(* CODESYS project Command3.project

Project tree, tasks and I/O mapping:
  Device : CODESYS Control for Raspberry Pi SL, 3S - Smart Software Solutions GmbH, version 3.5.11.0
    application Application
      libraries: Standard, * (System); StringUtils, 3.5.11.0 (System); CoDeSys Memory Manager, 3.5.12.0 (3S - Smart Software Solutions GmbH)
      task Task (cyclic, interval t#20ms, priority 1) calls MAIN
      POUs/
        Commands/
          function block FB_SocketOffCommand [ST]: Execute, FB_init, Undo
          function block FB_AirConComfortCommand [ST]: Execute, FB_init, Undo
          function block FB_AirConStandbyCommand [ST]: Execute, FB_init, Undo
          function block FB_SocketOnCommand [ST]: Execute, FB_init, Undo
          function block FB_LampSetLevelCommand [ST]: Execute, FB_init, Undo
          function block FB_MusicPlayCommand [ST]: Execute, FB_init, Undo
          function block FB_MusicStopCommand [ST]: Undo, Execute, FB_init
          interface I_Command: Execute, Undo
        Receiver/
          function block FB_Socket [ST]: Active, Off, On
          function block FB_Lamp [ST]: SetLevel, Level
          function block FB_CDPlayer [ST]: Volume, SetTrack, SetVolume, Start, Stop, PlayerActive, Track
          function block FB_AirConditioning [ST]: Activate, Deactivate, SetTemperature, Activated, Temperature
        Invoker/
          function block FB_SwitchPanel [ST]: FB_init, SetCommand
        program MAIN [ST]
    SoftMotion General Axis Pool
    I²C
    SPI
    GPIOs_A_B : GPIOs A/B, 3S - Smart Software Solutions GmbH, version 3.5.11.0
        unmapped channels: digital inputs (GPIO0..GPIO31), digital outputs (GPIO0..GPIO31)
    Onewire
    Camera device
      <Empty>
*)

// Device/Application/POUs/MAIN
PROGRAM MAIN
VAR
	// Invoker
	fbSwitchPanel				: FB_SwitchPanel;
	
	// Receiver
	fbSocket					: FB_Socket;
	refSocket					: REFERENCE TO FB_Socket := fbSocket;	
	fbLamp						: FB_Lamp;
	refLamp						: REFERENCE TO FB_Lamp := fbLamp;	
	fbAirConditioning			: FB_AirConditioning;
	refAirConditioning			: REFERENCE TO FB_AirConditioning := fbAirConditioning;
	fbCDPlayer					: FB_CDPlayer;
	refCDPlayer					: REFERENCE TO FB_CDPlayer := fbCDPlayer;

	// Commands
	fbSocketOnCommand			: FB_SocketOnCommand(refSocket);
	fbSocketOffCommand			: FB_SocketOffCommand(refSocket);
	fbLampSetLevel100Command	: FB_LampSetLevelCommand(refLamp, 100);
	fbLampSetLevel0Command		: FB_LampSetLevelCommand(refLamp, 0);
	fbAirConComfortCommand		: FB_AirConComfortCommand(refAirConditioning);
	fbAirConStandbyCommand		: FB_AirConStandbyCommand(refAirConditioning);	
	fbMusicPlayCommand			: FB_MusicPlayCommand(refCDPlayer);
	fbMusicStopCommand			: FB_MusicStopCommand(refCDPlayer);
	bInit						      : BOOL := TRUE;	
END_VAR

IF bInit THEN
	fbSwitchPanel.SetCommand(1, fbSocketOnCommand);
	fbSwitchPanel.SetCommand(2, fbSocketOffCommand);
	fbSwitchPanel.SetCommand(3, fbLampSetLevel100Command);
	fbSwitchPanel.SetCommand(4, fbLampSetLevel0Command);
	fbSwitchPanel.SetCommand(5, fbAirConComfortCommand);
	fbSwitchPanel.SetCommand(6, fbAirConStandbyCommand);
	fbSwitchPanel.SetCommand(7, fbMusicPlayCommand);
	fbSwitchPanel.SetCommand(8, fbMusicStopCommand);
	bInit := FALSE;;
ELSE
	fbSwitchPanel();	
END_IF

END_PROGRAM

// Device/Application/POUs/Invoker/FB_SwitchPanel
FUNCTION_BLOCK PUBLIC FB_SwitchPanel
VAR_INPUT
	bUndo			: BOOL;
	arrSwitch		: ARRAY[1..8] OF BOOL;
END_VAR
VAR
	aiCommand		: ARRAY[1..8] OF I_Command;	
	arrRtrig		: ARRAY[1..8] OF R_TRIG;
	iLastCommand	: I_Command;
	fbRtrigUndo		: R_TRIG;
	nIndex			: INT;
END_VAR

FOR nIndex := 1 TO 8 DO
	arrRtrig[nIndex](CLK := arrSwitch[nIndex]);
	IF arrRtrig[nIndex].Q THEN
		IF (aiCommand[nIndex] <> 0) THEN
			aiCommand[nIndex].Execute();
			iLastCommand := aiCommand[nIndex];
		END_IF
	END_IF
END_FOR

fbRtrigUndo(CLK := bUndo);
IF fbRtrigUndo.Q THEN
	IF (iLastCommand <> 0) THEN
		iLastCommand.Undo();
	END_IF
END_IF

METHOD FB_init : BOOL
VAR_INPUT
	bInitRetains : BOOL; // if TRUE, the retain variables are initialized (warm start / cold start)
	bInCopyCode : BOOL;  // if TRUE, the instance afterwards gets moved into the copy code (online change)
END_VAR
VAR
	nIndex : INT;
END_VAR
FOR nIndex := 1 TO 8 DO
	aiCommand[nIndex] := 0;
END_FOR
iLastCommand := 0;
END_METHOD

METHOD PUBLIC SetCommand : BOOL
VAR_INPUT
	nPosition		: INT;
	iCommand		: I_Command;
END_VAR
IF ((nPosition >= 1) AND (nPosition <= 8) AND (iCommand <> 0)) THEN
	THIS^.aiCommand[nPosition] := iCommand;
END_IF
END_METHOD

END_FUNCTION_BLOCK

// Device/Application/POUs/Commands/I_Command
INTERFACE I_Command

METHOD Execute
END_METHOD

METHOD Undo
END_METHOD

END_INTERFACE

// Device/Application/POUs/Receiver/FB_Socket
FUNCTION_BLOCK PUBLIC FB_Socket
VAR_OUTPUT
	bActive		: BOOL;
END_VAR

PROPERTY PUBLIC Active : BOOL
GET
Active := bActive;
END_GET
END_PROPERTY

METHOD PUBLIC Off
bActive := false;
END_METHOD

METHOD PUBLIC On
bActive := true;
END_METHOD

END_FUNCTION_BLOCK

// Device/Application/POUs/Receiver/FB_Lamp
FUNCTION_BLOCK PUBLIC FB_Lamp
VAR_OUTPUT
	byLevel			: BYTE;
END_VAR

METHOD PUBLIC SetLevel : BOOL
VAR_INPUT
	byNewLevel			: BYTE;
END_VAR
byLevel := byNewLevel;
END_METHOD

PROPERTY PUBLIC Level : BYTE
GET
Level := byLevel;
END_GET
END_PROPERTY

END_FUNCTION_BLOCK

// Device/Application/POUs/Receiver/FB_AirConditioning
FUNCTION_BLOCK PUBLIC FB_AirConditioning
VAR_OUTPUT
	bActive			: BOOL;
	lrTemperature	: LREAL;
END_VAR

METHOD PUBLIC Activate
bActive := TRUE;
END_METHOD

METHOD PUBLIC Deactivate
bActive := false;
END_METHOD

METHOD PUBLIC SetTemperature : BOOL
VAR_INPUT
	lrNewTemperature	: LREAL;
END_VAR
lrTemperature := lrNewTemperature;
END_METHOD

PROPERTY PUBLIC Activated : BOOL
GET
Activated := bActive;
END_GET
END_PROPERTY

PROPERTY PUBLIC Temperature : LREAL
GET
Temperature := lrTemperature;
END_GET
END_PROPERTY

END_FUNCTION_BLOCK

// Device/Application/POUs/Receiver/FB_CDPlayer
FUNCTION_BLOCK PUBLIC FB_CDPlayer
VAR_OUTPUT
	bPlayerActive		: BOOL;
	byVolume			: BYTE;
	byTrack				: UINT;
END_VAR

PROPERTY PUBLIC Volume : BYTE
GET
Volume := byVolume;
END_GET
END_PROPERTY

METHOD PUBLIC SetTrack : BOOL
VAR_INPUT
	byNewTrack			: UINT;
END_VAR
byTrack := byNewTrack;
END_METHOD

METHOD PUBLIC SetVolume : BOOL
VAR_INPUT
	byNewVolume 		: BYTE;
END_VAR
byVolume := byNewVolume;
END_METHOD

METHOD PUBLIC Start
bPlayerActive := true;
END_METHOD

METHOD PUBLIC Stop
bPlayerActive := FALSE;
END_METHOD

PROPERTY PUBLIC PlayerActive : BOOL
GET
PlayerActive := bPlayerActive;
END_GET
END_PROPERTY

PROPERTY PUBLIC Track : UINT
GET
Track := byTrack;
END_GET
END_PROPERTY

END_FUNCTION_BLOCK

// Device/Application/POUs/Commands/FB_SocketOnCommand
FUNCTION_BLOCK PUBLIC FB_SocketOnCommand IMPLEMENTS I_Command
VAR
	refSocket : REFERENCE TO FB_Socket;
END_VAR

METHOD Execute
IF (__ISVALIDREF(THIS^.refSocket)) THEN
	THIS^.refSocket.On();
END_IF
END_METHOD

METHOD FB_init : BOOL
VAR_INPUT
	bInitRetains : BOOL; // if TRUE, the retain variables are initialized (warm start / cold start)
	bInCopyCode : BOOL;  // if TRUE, the instance afterwards gets moved into the copy code (online change)
	refNewSocket : REFERENCE TO FB_Socket;
END_VAR
IF (__ISVALIDREF(refNewSocket)) THEN
	THIS^.refSocket REF= refNewSocket;
ELSE
	THIS^.refSocket REF= 0;
END_IF
END_METHOD

METHOD Undo
IF (__ISVALIDREF(THIS^.refSocket)) THEN
	THIS^.refSocket.Off();
END_IF
END_METHOD

END_FUNCTION_BLOCK

// Device/Application/POUs/Commands/FB_SocketOffCommand
FUNCTION_BLOCK PUBLIC FB_SocketOffCommand IMPLEMENTS I_Command
VAR
	refSocket : REFERENCE TO FB_Socket;
END_VAR

METHOD Execute
IF (__ISVALIDREF(THIS^.refSocket)) THEN
	THIS^.refSocket.Off();
END_IF
END_METHOD

METHOD FB_init : BOOL
VAR_INPUT
	bInitRetains : BOOL; // if TRUE, the retain variables are initialized (warm start / cold start)
	bInCopyCode : BOOL;  // if TRUE, the instance afterwards gets moved into the copy code (online change)
	refNewSocket : REFERENCE TO FB_Socket;
END_VAR
IF (__ISVALIDREF(refNewSocket)) THEN
	THIS^.refSocket REF= refNewSocket;
ELSE
	THIS^.refSocket REF= 0;
END_IF
END_METHOD

METHOD Undo
IF (__ISVALIDREF(THIS^.refSocket)) THEN
	THIS^.refSocket.On();
END_IF
END_METHOD

END_FUNCTION_BLOCK

// Device/Application/POUs/Commands/FB_LampSetLevelCommand
FUNCTION_BLOCK PUBLIC FB_LampSetLevelCommand IMPLEMENTS I_Command
VAR
	refLamp		: REFERENCE TO FB_Lamp;
	byNewLevel	: BYTE;
	byLastLevel : BYTE := 255;
END_VAR

METHOD Execute
IF (__ISVALIDREF(THIS^.refLamp)) THEN
	THIS^.byLastLevel := THIS^.refLamp.Level;	
	THIS^.refLamp.SetLevel(THIS^.byNewLevel);
END_IF
END_METHOD

METHOD FB_init : BOOL
VAR_INPUT
	bInitRetains : BOOL; // if TRUE, the retain variables are initialized (warm start / cold start)
	bInCopyCode : BOOL;  // if TRUE, the instance afterwards gets moved into the copy code (online change)
	refLamp : REFERENCE TO FB_Lamp;
	byNewLevel : BYTE;
END_VAR
IF (__ISVALIDREF(refLamp)) THEN
	THIS^.refLamp REF= refLamp;
ELSE
	THIS^.refLamp REF= 0;
END_IF
THIS^.byNewLevel := byNewLevel;
END_METHOD

METHOD Undo
IF (__ISVALIDREF(THIS^.refLamp)) THEN
	IF (THIS^.byLastLevel <> 255) THEN
		THIS^.refLamp.SetLevel(THIS^.byLastLevel);
	END_IF
END_IF
END_METHOD

END_FUNCTION_BLOCK

// Device/Application/POUs/Commands/FB_AirConComfortCommand
FUNCTION_BLOCK PUBLIC FB_AirConComfortCommand IMPLEMENTS I_Command
VAR
	refAirConditioning : REFERENCE TO FB_AirConditioning;
END_VAR

METHOD Execute
IF (__ISVALIDREF(THIS^.refAirConditioning)) THEN
	THIS^.refAirConditioning.Activate();
	THIS^.refAirConditioning.SetTemperature(20.0);
END_IF
END_METHOD

METHOD FB_init : BOOL
VAR_INPUT
	bInitRetains : BOOL; // if TRUE, the retain variables are initialized (warm start / cold start)
	bInCopyCode : BOOL;  // if TRUE, the instance afterwards gets moved into the copy code (online change)
	refAirConditioning : REFERENCE TO FB_AirConditioning;
END_VAR
IF (__ISVALIDREF(refAirConditioning)) THEN
	THIS^.refAirConditioning REF= refAirConditioning;
ELSE
	THIS^.refAirConditioning REF= 0;
END_IF
END_METHOD

METHOD Undo
IF (__ISVALIDREF(THIS^.refAirConditioning)) THEN
	THIS^.refAirConditioning.Activate();
	THIS^.refAirConditioning.SetTemperature(17.5);
END_IF
END_METHOD

END_FUNCTION_BLOCK

// Device/Application/POUs/Commands/FB_AirConStandbyCommand
FUNCTION_BLOCK PUBLIC FB_AirConStandbyCommand IMPLEMENTS I_Command
VAR
	refAirConditioning : REFERENCE TO FB_AirConditioning;
END_VAR

METHOD Execute
IF (__ISVALIDREF(THIS^.refAirConditioning)) THEN
	THIS^.refAirConditioning.Activate();
	THIS^.refAirConditioning.SetTemperature(17.5);
END_IF
END_METHOD

METHOD FB_init : BOOL
VAR_INPUT
	bInitRetains : BOOL; // if TRUE, the retain variables are initialized (warm start / cold start)
	bInCopyCode : BOOL;  // if TRUE, the instance afterwards gets moved into the copy code (online change)
	refAirConditioning : REFERENCE TO FB_AirConditioning;
END_VAR
IF (__ISVALIDREF(refAirConditioning)) THEN
	THIS^.refAirConditioning REF= refAirConditioning;
ELSE
	THIS^.refAirConditioning REF= 0;
END_IF
END_METHOD

METHOD Undo
IF (__ISVALIDREF(THIS^.refAirConditioning)) THEN
	THIS^.refAirConditioning.Activate();
	THIS^.refAirConditioning.SetTemperature(20.0);
END_IF
END_METHOD

END_FUNCTION_BLOCK

// Device/Application/POUs/Commands/FB_MusicPlayCommand
FUNCTION_BLOCK PUBLIC FB_MusicPlayCommand IMPLEMENTS I_Command
VAR
	refCDPlayer : REFERENCE TO FB_CDPlayer;
END_VAR

METHOD Execute
IF (__ISVALIDREF(THIS^.refCDPlayer)) THEN
	THIS^.refCDPlayer.SetVolume(40);
	THIS^.refCDPlayer.SetTrack(1);
	THIS^.refCDPlayer.Start();
END_IF
END_METHOD

METHOD FB_init : BOOL
VAR_INPUT
	bInitRetains : BOOL; // if TRUE, the retain variables are initialized (warm start / cold start)
	bInCopyCode : BOOL;  // if TRUE, the instance afterwards gets moved into the copy code (online change)
	refCDPlayer : REFERENCE TO FB_CDPlayer;
END_VAR
IF (__ISVALIDREF(refCDPlayer)) THEN
	THIS^.refCDPlayer REF= refCDPlayer;
ELSE
	THIS^.refCDPlayer REF= 0;
END_IF
END_METHOD

METHOD Undo
IF (__ISVALIDREF(THIS^.refCDPlayer)) THEN
	THIS^.refCDPlayer.Stop();
END_IF
END_METHOD

END_FUNCTION_BLOCK

// Device/Application/POUs/Commands/FB_MusicStopCommand
FUNCTION_BLOCK PUBLIC FB_MusicStopCommand IMPLEMENTS I_Command
VAR
	refCDPlayer : REFERENCE TO FB_CDPlayer;
END_VAR

METHOD Undo
IF (__ISVALIDREF(THIS^.refCDPlayer)) THEN
	THIS^.refCDPlayer.SetVolume(40);
	THIS^.refCDPlayer.SetTrack(1);
	THIS^.refCDPlayer.Start();
END_IF
END_METHOD

METHOD Execute
IF (__ISVALIDREF(THIS^.refCDPlayer)) THEN
	THIS^.refCDPlayer.Stop();
END_IF
END_METHOD

METHOD FB_init : BOOL
VAR_INPUT
	bInitRetains : BOOL; // if TRUE, the retain variables are initialized (warm start / cold start)
	bInCopyCode : BOOL;  // if TRUE, the instance afterwards gets moved into the copy code (online change)
	refCDPlayer : REFERENCE TO FB_CDPlayer;
END_VAR
IF (__ISVALIDREF(refCDPlayer)) THEN
	THIS^.refCDPlayer REF= refCDPlayer;
ELSE
	THIS^.refCDPlayer REF= 0;
END_IF
END_METHOD

END_FUNCTION_BLOCK
